PROGRAM pouMsgS2
VAR
	
	
	
END_VAR

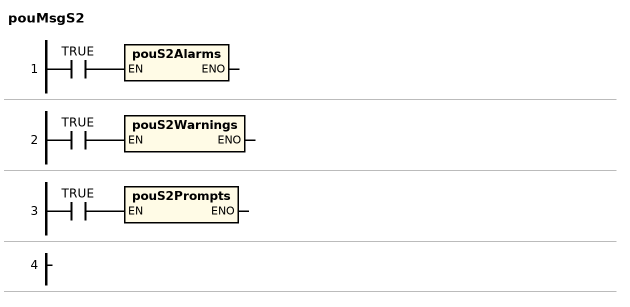
// NETWORK 1
pouS2Alarms();

// NETWORK 2
pouS2Warnings();

// NETWORK 3
pouS2Prompts();

// NETWORK 4

END_PROGRAM

(* stored: Version 1.1.0.1, ProductVersion 3.1.4024.12
   POU pouMsgS2: Id {c7604588-1c1b-47fa-a7a9-b4a5e6439762}, SpecialFunc None *)
